{attribute addProperty BoxType "EL3314-0002-0016"}
{attribute addProperty Id "TC_Inputs_ChannelAT %I*ARRAY[0..3] OF TC_Inputs_Channel_5C824630192240WcStateAT %I*WcState_98A4DF7520.250InfoDataAT %I*InfoData_BC63D37F80100"}
{attribute addProperty CRC "849042189"}
{attribute addProperty SizeInBites "274"}
{attribute addProperty SizeInBytes "34.25"}
TYPE EL3314_BFD35287 :
STRUCT
	{attribute addProperty Name "TC_Inputs_Channel"}
	TC_Inputs_Channel : ARRAY[0..3] OF TC_Inputs_Channel_5C824630;
	{attribute addProperty Name "WcState"}
	WcState : WcState_98A4DF75;
	{attribute addProperty Name "InfoData"}
	InfoData : InfoData_BC63D37F;
END_STRUCT
END_TYPE

(* stored: Version 1.2.0.0, ProductVersion 3.1.4024.9
   DUT EL3314_BFD35287: Id {4dbbd4c6-e0b6-44e1-ab29-065ec7a8f7b5} *)
